// SIMATIC S7-200 project (STEP 7-Micro/WIN), CPU 224XP REL 02.01

SYMBOL_TABLE USUARIO1
P_PARO           I0.0
P_DERECHAS       I0.1
P_IZQUIERDAS     I0.2
RELE_TERMICO     I0.4
LED_PARO         Q0.0
L_DERECHAS       Q0.1
L_IZQUIERDAS     Q0.2
ESTRELLA         Q0.3
TRIANGULO        Q0.4
LED_DERECHAS     Q0.5
LED_IZQUIERDAS   Q0.6
LED_AVERIA       Q0.7
END_SYMBOL_TABLE

ORGANIZATION_BLOCK PRINCIPAL:OB1
TITLE=COMENTARIOS DEL PROGRAMA
BEGIN
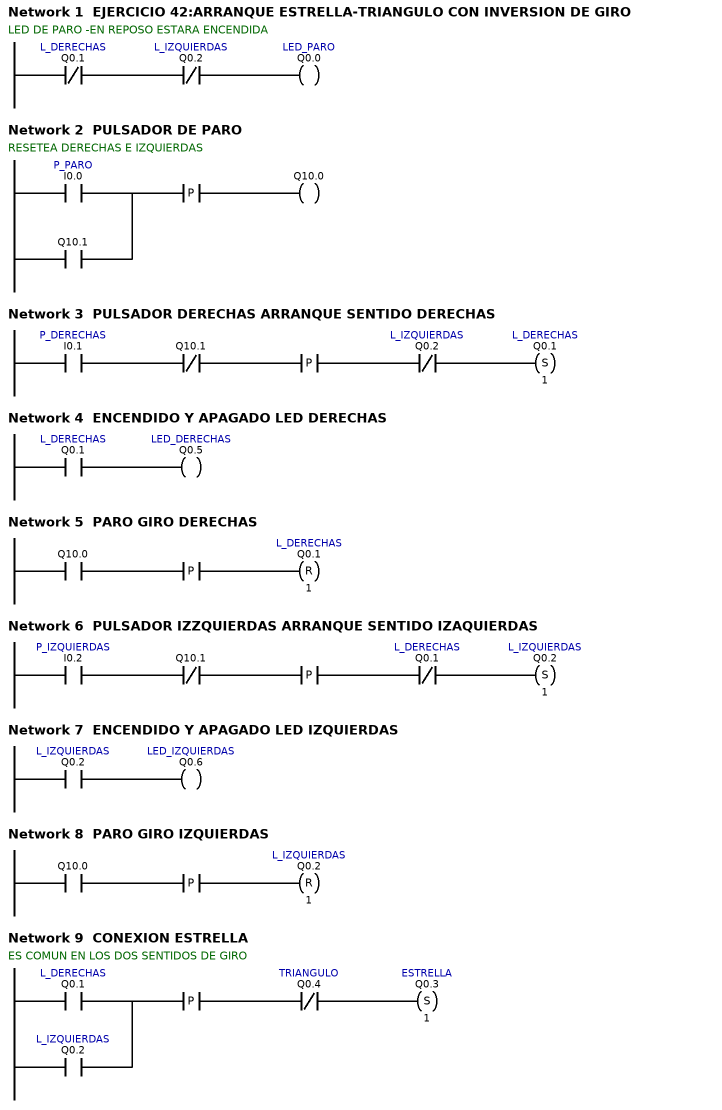
Network 1 // EJERCICIO 42:ARRANQUE ESTRELLA-TRIANGULO CON INVERSION DE GIRO
// LED DE PARO -EN REPOSO ESTARA ENCENDIDA
LDN    L_DERECHAS:Q0.1
AN     L_IZQUIERDAS:Q0.2
=      LED_PARO:Q0.0
Network 2 // PULSADOR DE PARO
// RESETEA DERECHAS E IZQUIERDAS
LD     P_PARO:I0.0
O      Q10.1
EU
=      Q10.0
Network 3 // PULSADOR DERECHAS ARRANQUE SENTIDO DERECHAS
LD     P_DERECHAS:I0.1
AN     Q10.1
EU
AN     L_IZQUIERDAS:Q0.2
S      L_DERECHAS:Q0.1, 1
Network 4 // ENCENDIDO Y APAGADO LED DERECHAS
LD     L_DERECHAS:Q0.1
=      LED_DERECHAS:Q0.5
Network 5 // PARO GIRO DERECHAS
LD     Q10.0
EU
R      L_DERECHAS:Q0.1, 1
Network 6 // PULSADOR IZZQUIERDAS ARRANQUE SENTIDO IZAQUIERDAS
LD     P_IZQUIERDAS:I0.2
AN     Q10.1
EU
AN     L_DERECHAS:Q0.1
S      L_IZQUIERDAS:Q0.2, 1
Network 7 // ENCENDIDO Y APAGADO LED IZQUIERDAS
LD     L_IZQUIERDAS:Q0.2
=      LED_IZQUIERDAS:Q0.6
Network 8 // PARO GIRO IZQUIERDAS
LD     Q10.0
EU
R      L_IZQUIERDAS:Q0.2, 1
Network 9 // CONEXION ESTRELLA
// ES COMUN EN LOS DOS SENTIDOS DE GIRO
LD     L_DERECHAS:Q0.1
O      L_IZQUIERDAS:Q0.2
EU
AN     TRIANGULO:Q0.4
S      ESTRELLA:Q0.3, 1
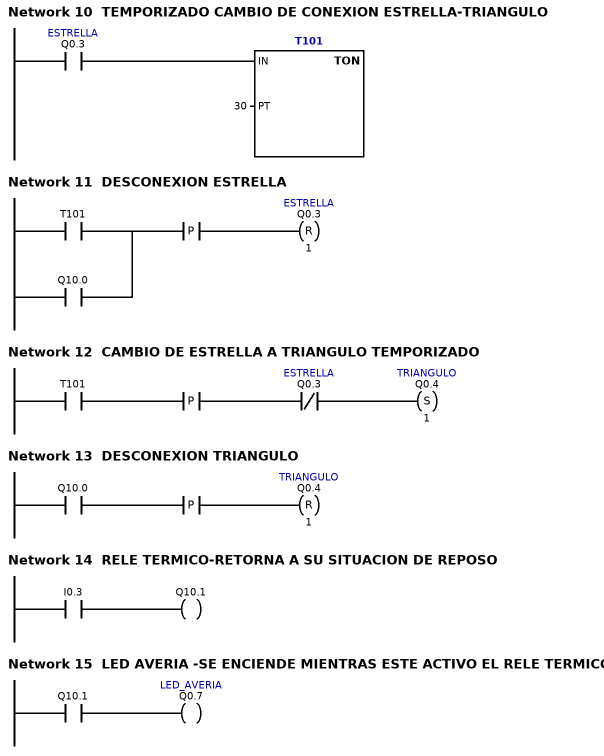
Network 10 // TEMPORIZADO CAMBIO DE CONEXION ESTRELLA-TRIANGULO
LD     ESTRELLA:Q0.3
TON    T101, 30
Network 11 // DESCONEXION ESTRELLA
LD     T101
O      Q10.0
EU
R      ESTRELLA:Q0.3, 1
Network 12 // CAMBIO DE ESTRELLA A TRIANGULO TEMPORIZADO
LD     T101
EU
AN     ESTRELLA:Q0.3
S      TRIANGULO:Q0.4, 1
Network 13 // DESCONEXION TRIANGULO
LD     Q10.0
EU
R      TRIANGULO:Q0.4, 1
Network 14 // RELE TERMICO-RETORNA A SU SITUACION DE REPOSO
LD     I0.3
=      Q10.1
Network 15 // LED AVERIA -SE ENCIENDE MIENTRAS ESTE ACTIVO EL RELE TERMICO
LD     Q10.1
=      LED_AVERIA:Q0.7
END_ORGANIZATION_BLOCK
